{attribute 'linkalways'} 
{attribute 'no_explicit_call' := 'This FB is a CLASS and must be accessed using methods or properties'}
{attribute 'enable_dynamic_creation'}
FUNCTION_BLOCK _ETcVnDiffusivityTypeKAZE EXTENDS EnumDatatypeBase
VAR
	localData : ETcVnDiffusivityTypeKAZE;
	activeData : REFERENCE TO ETcVnDiffusivityTypeKAZE;
	enumBaseDatatype : _DINT(localData);
END_VAR

METHOD PRIVATE AddLocalEnumeration
VAR_INPUT
	Enumeration : T_MAXSTRING;
	Value : ETcVnDiffusivityTypeKAZE;
END_VAR
AddEnumeration(Enumeration, Value);
END_METHOD

PROPERTY PUBLIC Address : PVOID
GET
Address := ADR(activeData);
END_GET
END_PROPERTY

METHOD PUBLIC ClearReference
VAR_INPUT
END_VAR
activeData REF= localData;
SetBaseDatatypeReference();
END_METHOD

METHOD PUBLIC Clone : I_Datatype
VAR
    pClone : POINTER TO _ETcVnDiffusivityTypeKAZE;
END_VAR
pClone := __NEW(_ETcVnDiffusivityTypeKAZE(InitialValue := Value));
Clone := pClone^;
END_METHOD

METHOD FB_init : BOOL
VAR_INPUT
	bInitRetains : BOOL; // if TRUE, the retain variables are initialized (warm start / cold start)
	bInCopyCode : BOOL;  // if TRUE, the instance afterwards gets moved into the copy code (online change)
	InitialValue : ETcVnDiffusivityTypeKAZE;
END_VAR
localData := InitialValue;
AddBaseDatatype(enumBaseDatatype);
ClearReference();

AddLocalEnumeration('TCVN_DT1_KAZE_PM_G1', ETcVnDiffusivityTypeKAZE.TCVN_DT1_KAZE_PM_G1);
AddLocalEnumeration('TCVN_DT1_KAZE_PM_G2', ETcVnDiffusivityTypeKAZE.TCVN_DT1_KAZE_PM_G2);
AddLocalEnumeration('TCVN_DT1_KAZE_WEICKERT', ETcVnDiffusivityTypeKAZE.TCVN_DT1_KAZE_WEICKERT);
AddLocalEnumeration('TCVN_DT1_KAZE_CHARBONNIER', ETcVnDiffusivityTypeKAZE.TCVN_DT1_KAZE_CHARBONNIER);
END_METHOD

PROPERTY PUBLIC Identifier : T_MAXSTRING
GET
Identifier := 'ETcVnDiffusivityTypeKAZE';
END_GET
END_PROPERTY

METHOD IsEnumeratorValueEqual : BOOL
VAR_INPUT
	Enumerator : I_KeyValueForwardEnumerator;
END_VAR
VAR
	storedValue : ETcVnDiffusivityTypeKAZE;
END_VAR
IF NOT Enumerator.TryGet(storedValue) THEN
	RETURN;
END_IF

IsEnumeratorValueEqual := storedValue = activeData;
END_METHOD

METHOD PUBLIC MakeReferenceTo
VAR_INPUT
	ReferenceTarget : REFERENCE TO ETcVnDiffusivityTypeKAZE;
END_VAR
activeData REF= ReferenceTarget;
SetBaseDatatypeReference();
END_METHOD

METHOD PROTECTED SetBaseDatatypeReference
VAR_INPUT
END_VAR
enumBaseDatatype.MakeReferenceTo(activeData);
END_METHOD

PROPERTY PUBLIC Size : UDINT
GET
Size := SIZEOF(activeData);
END_GET
END_PROPERTY

METHOD TryMakeReferenceTo : BOOL
VAR_INPUT
	Target : I_Datatype;
END_VAR
VAR
	targetAsEnum : I_EnumDatatype;
	pTargetData : POINTER TO ETcVnDiffusivityTypeKAZE;
END_VAR
IF NOT Target.TryResolveAsEnumDatatype(targetAsEnum) THEN
	RETURN;
END_IF

IF targetAsEnum.Identifier <> Identifier THEN
	RETURN;
END_IF

pTargetData := Target.Address;
activeData REF= pTargetData^;
SetBaseDatatypeReference();
TryMakeReferenceTo := TRUE;
END_METHOD

PROPERTY PUBLIC Value : ETcVnDiffusivityTypeKAZE
GET
Value := activeData;
END_GET
SET
activeData := Value;
END_SET
END_PROPERTY

END_FUNCTION_BLOCK

(* stored: Version 1.1.0.1
   POU _ETcVnDiffusivityTypeKAZE: Id {ff3477bf-acc1-441e-b815-b5c3f507eea9}, SpecialFunc None
   Folder Constructor: Id {f136d775-00ba-4d47-b8b8-f062c471fe79}
   Folder Private: Id {dea3cdec-7b76-43fb-b6a9-c2e730e7db5d}
   Folder Protected: Id {8964923b-2c8b-4b86-bf6e-9bf252b2a03e}
   Method AddLocalEnumeration: Id {a23e9b24-d759-4f3b-9fd2-c1f08d68957a}
   Property Address: Id {14205042-54b2-454e-a859-a1409e9110fc}
   Get Get: Id {38e2f660-9e65-4583-9cf3-f125d9e84d4b}
   Method ClearReference: Id {3ec39f8c-0d70-4597-86ea-47b0034b7866}
   Method Clone: Id {5ca324fd-11e9-4048-b71e-25880fef5ffc}
   Method FB_init: Id {03734ee1-d59c-4423-8e3e-b722d25eb47a}
   Property Identifier: Id {6297a846-8d8f-4be9-a526-3e64a16a47da}
   Get Get: Id {d2e2ccc3-c5a2-4b9d-93c5-1b81117f13a1}
   Method IsEnumeratorValueEqual: Id {8db897ea-b113-448d-8550-1d744acd06e9}
   Method MakeReferenceTo: Id {a444450e-88e2-48cd-8dfb-9cef9a89b4e2}
   Method SetBaseDatatypeReference: Id {a28752f2-a78d-4ce2-a1e8-f3f0c110edc3}
   Property Size: Id {b210f3e0-b23e-4e90-8c46-b30cdeba26d8}
   Get Get: Id {9aaaed6b-3a6a-4ddd-a1b4-ad4e5d78cfc7}
   Method TryMakeReferenceTo: Id {0764a77d-4ff2-428d-a416-25d1a2d2ff2f}
   Property Value: Id {84b12e9a-c139-4907-85ff-cbd19494452a}
   Get Get: Id {4133a307-b20d-4e64-a657-384648206a19}
   Set Set: Id {7a80dadb-8833-452d-b054-4f56ffdb89c3} *)
